(* IEC 61131-3 sources: Industry-PLC-LLM/data/PLCBEAD_repo/PLCBEAD_PLCEmbed-main/PLC-BEAD/Source/GEB/RANGE_TO_WORD, 1 file *)

(* ---- RANGE_TO_WORD.ST ---- *)
FUNCTION TRUNC_REAL:REAL

	VAR_INPUT
		IN :	REAL;
	END_VAR

	TRUNC_REAL := UDINT_TO_REAL(DINT_TO_UDINT(TRUNC(IN)));
END_FUNCTION

FUNCTION RANGE_TO_WORD:WORD

	VAR_INPUT
		X :	REAL;
		LOW :	REAL;
		HIGH :	REAL;
	END_VAR

	Range_to_Word := REAL_TO_WORD(TRUNC_REAL((LIMIT(low,X,high)-LOW) * 65535.0 / (HIGH - LOW)));

END_FUNCTION

PROGRAM program0

	VAR
		X :	REAL;
		LOW :	REAL;
		HIGH :	REAL;

        OUT :	WORD;
	END_VAR
	OUT := RANGE_TO_WORD(X, LOW, HIGH);

END_PROGRAM
